FUNCTION_BLOCK TEST_STARTPOINT
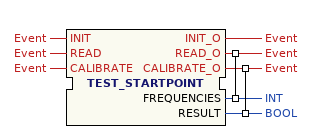
  EVENT_INPUT
    INIT;
    READ;
    CALIBRATE; {SET_ATTRIBUTE(OpcUa, Method)}
  END_EVENT
  EVENT_OUTPUT
    INIT_O;
    READ_O WITH FREQUENCIES;
    CALIBRATE_O WITH RESULT;
  END_EVENT
  VAR_OUTPUT
    FREQUENCIES : INT; {SET_ATTRIBUTE(OpcUa, Variable)}
    RESULT : BOOL; {SET_ATTRIBUTE(OpcUa, CALIBRATE)}
  END_VAR
END_FUNCTION_BLOCK
(* other elements stored in the file *)
(* SelfDescription FBType=POINT.STARTPOINT *)
